Staubli VAL3: sendAck.pgx

public program sendAck(sio& x_sSocket, num& x_nConnFlag, RosSimpleMsg& x_msg, num& x_nMsgRecvState)
begin
  // Copyright (c) 2016, Ocado Technology - Robotics Research Team
  // Copyright (c) 2021, Institute for Factory Automation and Production Systems (FAPS)
  //
  // Licensed under the Apache License, Version 2.0 (the "License");
  // you may not use this file except in compliance with the License.
  // You may obtain a copy of the License at
  //
  //     http://www.apache.org/licenses/LICENSE-2.0
  //
  // Unless required by applicable law or agreed to in writing, software
  // distributed under the License is distributed on an "AS IS" BASIS,
  // WITHOUT WARRANTIES OR CONDITIONS OF ANY KIND, either express or implied.
  // See the License for the specific language governing permissions and
  // limitations under the License.



  switch x_msg.header.nMsgType
    case SimpleMsg:MsgType.JOINT_TRAJ_PT
      call sendRosMsg(x_sSocket, rosTrajPtAck.prefix, rosTrajPtAck.header, rosTrajPtAck.body, x_nConnFlag)
    break
    case SimpleMsg:MsgType.JOINT_TRAJ_PT_F
      call sendRosMsg(x_sSocket, rosTrajPtFAck.prefix, rosTrajPtFAck.header, rosTrajPtFAck.body, x_nConnFlag)
    break
    // Staubli specific
    case Staubli:MsgType.SET_DRIVE_POWER
      call sendRosMsg(x_sSocket, Staubli:setDrvPwrAck.prefix, Staubli:setDrvPwrAck.header, Staubli:setDrvPwrAck.body, x_nConnFlag)
    break
    case Staubli:MsgType.WRITE_SINGLE_IO
      call sendRosMsg(x_sSocket, Staubli:writeSingIOAck.prefix, Staubli:writeSingIOAck.header, Staubli:writeSingIOAck.body, x_nConnFlag)
    break
    case Staubli:MsgType.VELOCITY_CFG
      call sendRosMsg(x_sSocket, Staubli:velCfgAck.prefix, Staubli:velCfgAck.header, Staubli:velCfgAck.body, x_nConnFlag)
    break
    case Staubli:MsgType.VELOCITY_CMD
      call sendRosMsg(x_sSocket, Staubli:velCmdAck.prefix, Staubli:velCmdAck.header, Staubli:velCmdAck.body, x_nConnFlag)
    break
    // default
    default
      //region @DEBUG
      if (bDebugMode and nDebugLevel<=5)
        call printDebug("sendAck: switch (msgType)",true)
        call printDebug("ERROR: unknown msg type",false)
      endIf
      //endregion
    break
  endSwitch

  // regardless of result from sending ACK
  // reset state machine to receive new messages
  x_nMsgRecvState = MsgRecvState.RECEIVE_HEADER
end
